TYPE FaultWarningState :
STRUCT
	IsActive :	BOOL;
END_STRUCT
END_TYPE

(* stored: Version 1.1.0.1
   DUT FaultWarningState: Id {ff6b7ca2-86e7-41b3-9ccc-196d939cd64e} *)
